{attribute 'qualified_only'}
{attribute 'strict'}
TYPE E_InverterState :
(
	Stopped 	:= 0,
	Starting 	:= 1,
	Started 	:= 2,
	Paused		:= 3,
	Stopping	:= 4,
	Alarm		:= 5
);
END_TYPE

(* stored: Version 1.1.0.1
   DUT E_InverterState: Id {48ebc780-4c00-40d2-963e-288b51d19fcf} *)
